// Mitsubishi GX Works2 project: BookEX6_40 String   PLC: Q13UDV

// global labels: Global
VAR_GLOBAL
  bVar0 AT M5000 : BOOL;
  abArray0 AT M5010 : ARRAY [0..49] OF BOOL;
  sStr0 AT D5000 : STRING[199];
  sStr1 AT D5100 : STRING[199];
  sStr2 AT D5200 : STRING[199];
  sStr3 AT D5300 : STRING[199];
  sStr4 AT D5400 : STRING[199];
  sStr5 AT D5500 : STRING[199];
  sStr6 AT D5600 : STRING[199];
  sStr7 AT D5700 : STRING[199];
  sStr8 AT D5800 : STRING[199];
  sStr9 AT D5900 : STRING[199];
  iVar0 AT D4500 : INT;
  iVar1 AT D4501 : INT;
  iVar2 AT D4502 : INT;
  iVar3 AT D4503 : INT;
  iVar4 AT D4504 : INT;
  iVar5 AT D4505 : INT;
  iVar6 AT D4506 : INT;
  iVar7 AT D4507 : INT;
  iVar8 AT D4508 : INT;
  iVar9 AT D4509 : INT;
  dVar0 AT D4510 : DINT;
  dVar1 AT D4512 : DINT;
  dVar2 AT D4514 : DINT;
  dVar3 AT D4516 : DINT;
  dVar4 AT D4518 : DINT;
  dVar5 AT D4520 : DINT;
  dVar6 AT D4522 : DINT;
  dVar7 AT D4524 : DINT;
  dVar8 AT D4526 : DINT;
  dVar9 AT D4528 : DINT;
  wVar0 AT D4530 : WORD;
  wVar1 AT D4531 : WORD;
  wVar2 AT D4532 : WORD;
  wVar3 AT D4533 : WORD;
  wVar4 AT D4534 : WORD;
  wVar5 AT D4535 : WORD;
  wVar6 AT D4536 : WORD;
  wVar7 AT D4537 : WORD;
  wVar8 AT D4538 : WORD;
  wVar9 AT D4539 : WORD;
  dwVar0 AT D4540 : DWORD;
  dwVar1 AT D4542 : DWORD;
  dwVar2 AT D4544 : DWORD;
  dwVar3 AT D4546 : DWORD;
  dwVar4 AT D4548 : DWORD;
  dwVar5 AT D4550 : DWORD;
  dwVar6 AT D4552 : DWORD;
  dwVar7 AT D4554 : DWORD;
  dwVar8 AT D4556 : DWORD;
  dwVar9 AT D4558 : DWORD;
  fsVar0 AT D4560 : REAL;
  fsVar1 AT D4562 : REAL;
  fsVar2 AT D4564 : REAL;
  fsVar3 AT D4566 : REAL;
  fsVar4 AT D4568 : REAL;
  fsVar5 AT D4570 : REAL;
  fsVar6 AT D4572 : REAL;
  fsVar7 AT D4574 : REAL;
  fsVar8 AT D4576 : REAL;
  fsVar9 AT D4578 : REAL;
  fdVar0 AT D4580 : LREAL;
  tTime0 AT D4620 : TIME;
  tTime1 AT D4622 : TIME;
  tTime2 AT D4624 : TIME;
  tTime3 AT D4626 : TIME;
  tTime4 AT D4628 : TIME;
  tTime5 AT D4630 : TIME;
  tTime6 AT D4632 : TIME;
  tTime7 AT D4634 : TIME;
  tTime8 AT D4636 : TIME;
  tTime9 AT D4638 : TIME;
  tTime10 AT D4640 : TIME;
  bVar1 AT M5001 : BOOL;
  bVar2 AT M5002 : BOOL;
  bVar3 AT M5003 : BOOL;
  bVar4 AT M5004 : BOOL;
  bVar5 AT M5005 : BOOL;
  bVar6 AT M5006 : BOOL;
  bVar7 AT M5007 : BOOL;
  bVar8 AT M5008 : BOOL;
  bVar9 AT M5009 : BOOL;
  abArray1 AT M5060 : ARRAY [0..49] OF BOOL;
  abArray2 AT M5110 : ARRAY [0..49] OF BOOL;
  abArray3 AT M5160 : ARRAY [0..49] OF BOOL;
  abArray4 AT M5210 : ARRAY [0..49] OF BOOL;
  abArray5 AT M5260 : ARRAY [0..49] OF BOOL;
  abArray6 AT M5310 : ARRAY [0..49] OF BOOL;
  abArray7 AT M5360 : ARRAY [0..49] OF BOOL;
  abArray8 AT M5410 : ARRAY [0..49] OF BOOL;
  abArray9 AT M5460 : ARRAY [0..49] OF BOOL;
  fdVar1 AT D4584 : LREAL;
  fdVar2 AT D4588 : LREAL;
  fdVar3 AT D4592 : LREAL;
  fdVar4 AT D4596 : LREAL;
  fdVar5 AT D4600 : LREAL;
  fdVar6 AT D4604 : LREAL;
  fdVar7 AT D4608 : LREAL;
  fdVar8 AT D4612 : LREAL;
  fdVar9 AT D4616 : LREAL;
  afsPen0 AT D2000 : ARRAY [0..499] OF REAL;
  afsPen1 AT D3000 : ARRAY [0..499] OF REAL;
  SpecStr AT D4999 : STRING[1];
  adwD10 AT D10 : ARRAY [0..9] OF DWORD;
  awD10 AT D10 : ARRAY [0..19] OF WORD;
  abM10 AT M10 : ARRAY [0..19] OF BOOL;
END_VAR
// user libraries (not included): HMI

PROGRAM ExASC_HEX
VAR
  Mov4WORD_1 : Mov4WORD;
  Mov4WORD_2 : Mov4WORD;
END_VAR
(* structured ladder/FBD written out as ST: instructions are called as NAME(EN, inputs, outputs); _pN, _eN, _tN stand for wires *)
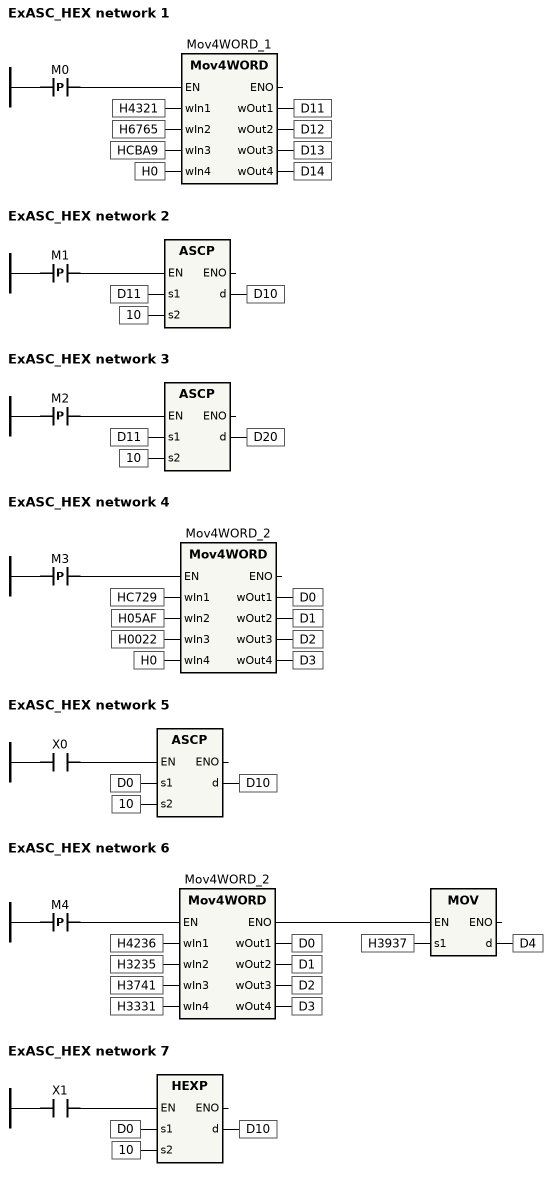
(* network 1 *)
Mov4WORD_1(EN := LDP(TRUE, M0), wIn1 := H4321, wIn2 := H6765, wIn3 := HCBA9, wIn4 := H0, wOut1 => D11, wOut2 => D12, wOut3 => D13, wOut4 => D14);
(* network 2 *)
ASCP(LDP(TRUE, M1), D11, 10, D10);
(* network 3 *)
ASCP(LDP(TRUE, M2), D11, 10, D20);
(* network 4 *)
Mov4WORD_2(EN := LDP(TRUE, M3), wIn1 := HC729, wIn2 := H05AF, wIn3 := H0022, wIn4 := H0, wOut1 => D0, wOut2 => D1, wOut3 => D2, wOut4 => D3);
(* network 5 *)
ASCP(X0, D0, 10, D10);
(* network 6 *)
Mov4WORD_2(EN := LDP(TRUE, M4), wIn1 := H4236, wIn2 := H3235, wIn3 := H3741, wIn4 := H3331, wOut1 => D0, wOut2 => D1, wOut3 => D2, wOut4 => D3);
MOV(Mov4WORD_2.ENO, H3937, D4);
(* network 7 *)
HEXP(X1, D0, 10, D10);
END_PROGRAM

PROGRAM ExBCDDA
VAR
  newBCDDA_1 : newBCDDA;
  sTemp : STRING[6];
END_VAR
(* structured ladder/FBD written out as ST: instructions are called as NAME(EN, inputs, outputs); _pN, _eN, _tN stand for wires *)
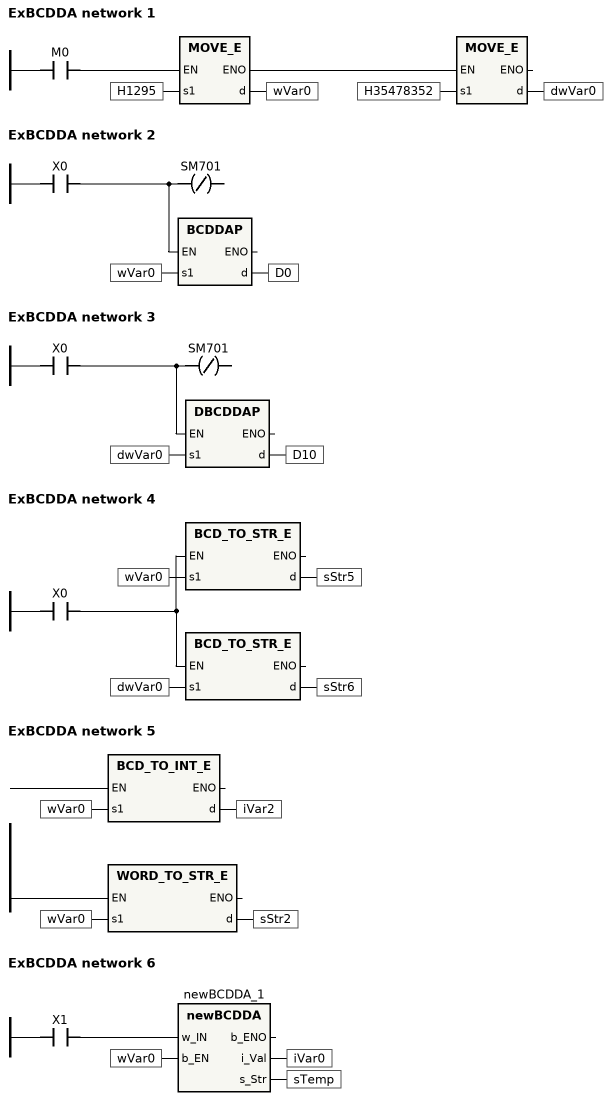
(* network 1 *)
_e1 := MOVE_E(M0, H1295, wVar0);
MOVE_E(_e1, H35478352, dwVar0);
(* network 2 *)
SM701 := NOT X0;
BCDDAP(X0, wVar0, D0);
(* network 3 *)
SM701 := NOT X0;
DBCDDAP(X0, dwVar0, D10);
(* network 4 *)
BCD_TO_STR_E(X0, wVar0, sStr5);
BCD_TO_STR_E(X0, dwVar0, sStr6);
(* network 5 *)
BCD_TO_INT_E(TRUE, wVar0, iVar2);
WORD_TO_STR_E(TRUE, wVar0, sStr2);
(* network 6 *)
newBCDDA_1(w_IN := X1, b_EN := wVar0, i_Val => iVar0, s_Str => sTemp);
END_PROGRAM

PROGRAM ExBINDA
(* structured ladder/FBD written out as ST: instructions are called as NAME(EN, inputs, outputs); _pN, _eN, _tN stand for wires *)
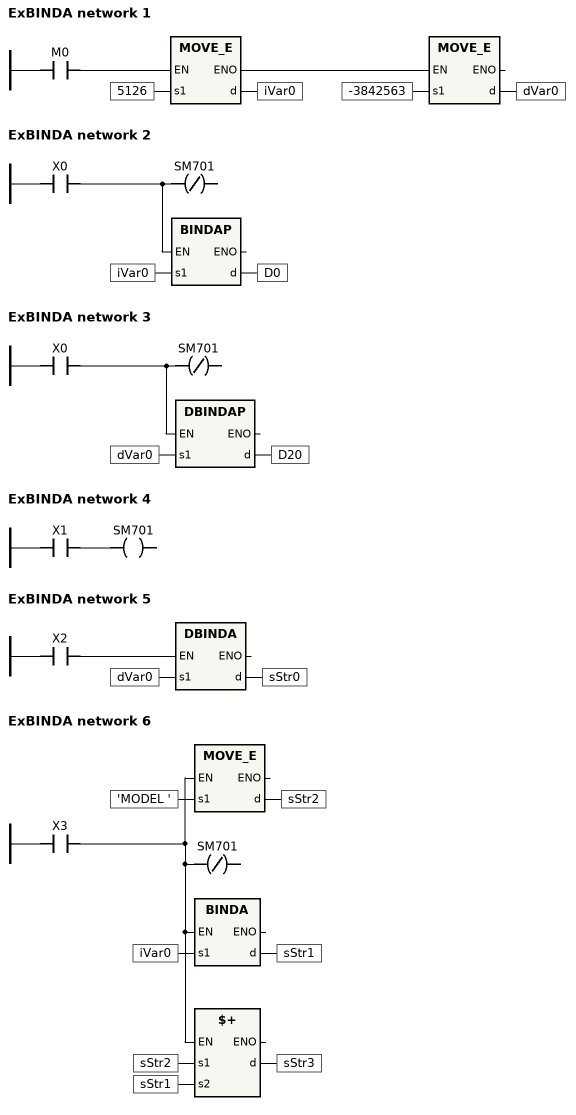
(* network 1 *)
_e1 := MOVE_E(M0, 5126, iVar0);
MOVE_E(_e1, -3842563, dVar0);
(* network 2 *)
SM701 := NOT X0;
BINDAP(X0, iVar0, D0);
(* network 3 *)
SM701 := NOT X0;
DBINDAP(X0, dVar0, D20);
(* network 4 *)
SM701 := X1;
(* network 5 *)
DBINDA(X2, dVar0, sStr0);
(* network 6 *)
SM701 := NOT X3;
MOVE_E(X3, 'MODEL ', sStr2);
BINDA(X3, iVar0, sStr1);
$+(X3, sStr2, sStr1, sStr3);
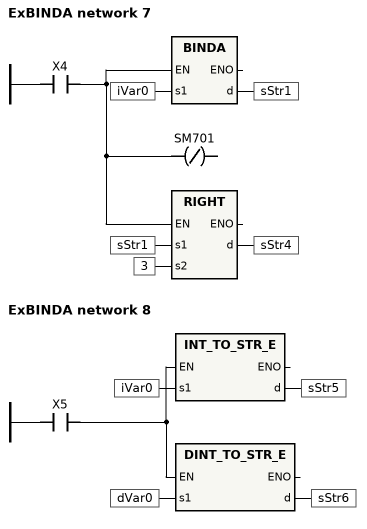
(* network 7 *)
SM701 := NOT X4;
BINDA(X4, iVar0, sStr1);
RIGHT(X4, sStr1, 3, sStr4);
(* network 8 *)
INT_TO_STR_E(X5, iVar0, sStr5);
DINT_TO_STR_E(X5, dVar0, sStr6);
END_PROGRAM

PROGRAM ExBINHA
VAR
  sStr40 : STRING[4];
  sStr41 : STRING[4];
END_VAR
(* structured ladder/FBD written out as ST: instructions are called as NAME(EN, inputs, outputs); _pN, _eN, _tN stand for wires *)
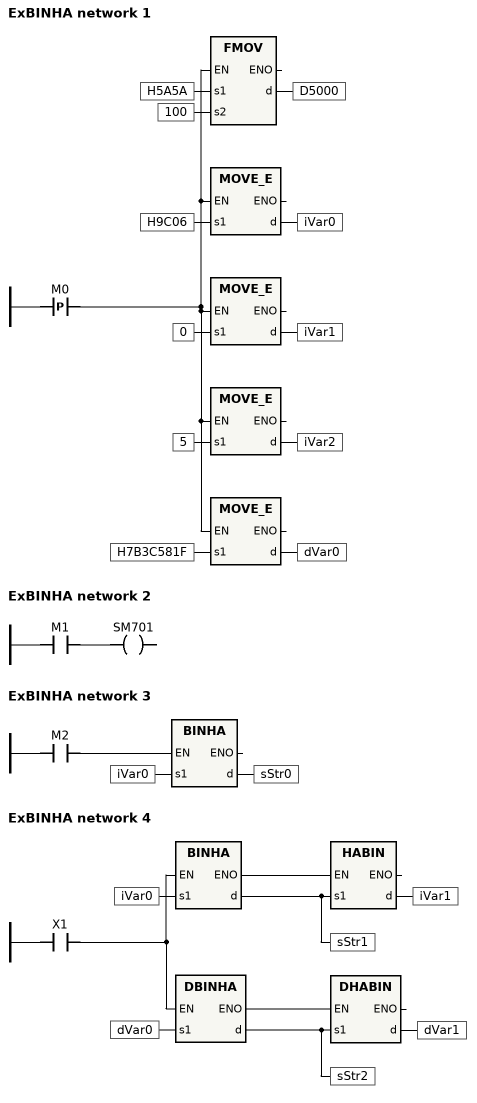
(* network 1 *)
_p1 := LDP(TRUE, M0);
FMOV(_p1, H5A5A, 100, D5000);
MOVE_E(_p1, H9C06, iVar0);
MOVE_E(_p1, 0, iVar1);
MOVE_E(_p1, 5, iVar2);
MOVE_E(_p1, H7B3C581F, dVar0);
(* network 2 *)
SM701 := M1;
(* network 3 *)
BINHA(M2, iVar0, sStr0);
(* network 4 *)
_e1 := BINHA(X1, iVar0, sStr1);
HABIN(_e1, sStr1, iVar1);
_e2 := DBINHA(X1, dVar0, sStr2);
DHABIN(_e2, sStr2, dVar1);
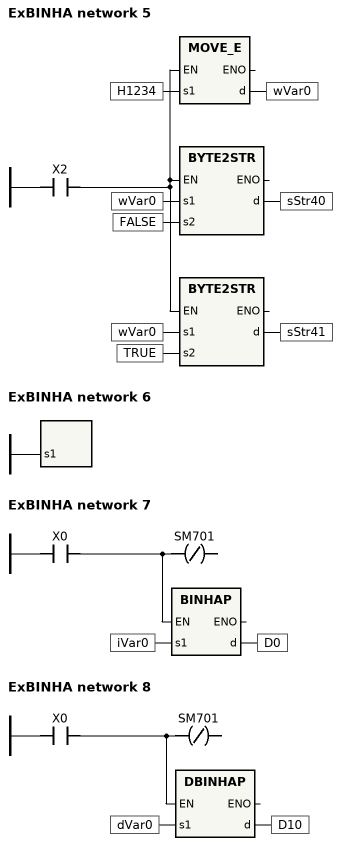
(* network 5 *)
MOVE_E(X2, H1234, wVar0);
BYTE2STR(X2, wVar0, FALSE, sStr40);
BYTE2STR(X2, wVar0, TRUE, sStr41);
(* network 6 *)
(* element kind 10  <- TRUE *)
(* network 7 *)
SM701 := NOT X0;
BINHAP(X0, iVar0, D0);
(* network 8 *)
SM701 := NOT X0;
DBINHAP(X0, dVar0, D10);
END_PROGRAM

PROGRAM ExCOMRD
VAR
  aiTmp : ARRAY [0..1] OF INT;
END_VAR
(* structured ladder/FBD written out as ST: instructions are called as NAME(EN, inputs, outputs); _pN, _eN, _tN stand for wires *)
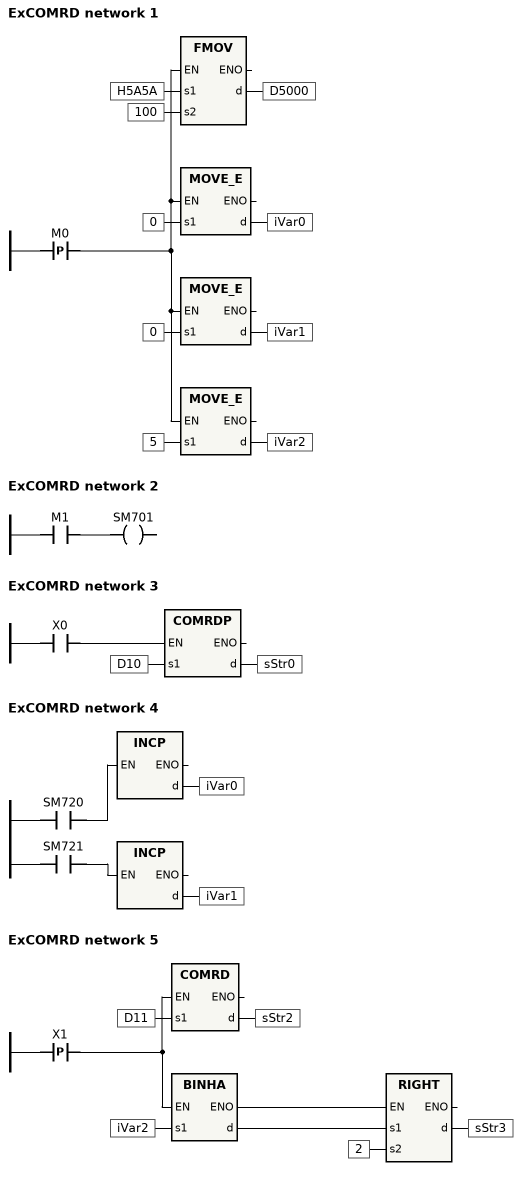
(* network 1 *)
_p1 := LDP(TRUE, M0);
FMOV(_p1, H5A5A, 100, D5000);
MOVE_E(_p1, 0, iVar0);
MOVE_E(_p1, 0, iVar1);
MOVE_E(_p1, 5, iVar2);
(* network 2 *)
SM701 := M1;
(* network 3 *)
COMRDP(X0, D10, sStr0);
(* network 4 *)
INCP(SM720, iVar0);
INCP(SM721, iVar1);
(* network 5 *)
_p1 := LDP(TRUE, X1);
COMRD(_p1, D11, sStr2);
_e3 := BINHA(_p1, iVar2, _t2);
RIGHT(_e3, _t2, 2, sStr3);
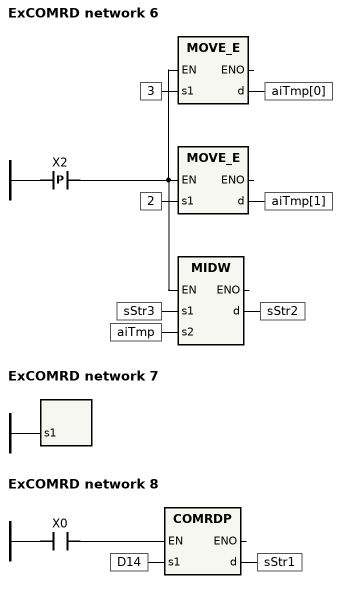
(* network 6 *)
_p1 := LDP(TRUE, X2);
MOVE_E(_p1, 3, aiTmp[0]);
MOVE_E(_p1, 2, aiTmp[1]);
MIDW(_p1, sStr3, aiTmp, sStr2);
(* network 7 *)
(* element kind 10  <- TRUE *)
(* network 8 *)
COMRDP(X0, D14, sStr1);
END_PROGRAM

PROGRAM ExDABCD
VAR
  UpperSTR_1 : UpperSTR;
  UpperSTR_2 : UpperSTR;
END_VAR
(* structured ladder/FBD written out as ST: instructions are called as NAME(EN, inputs, outputs); _pN, _eN, _tN stand for wires *)
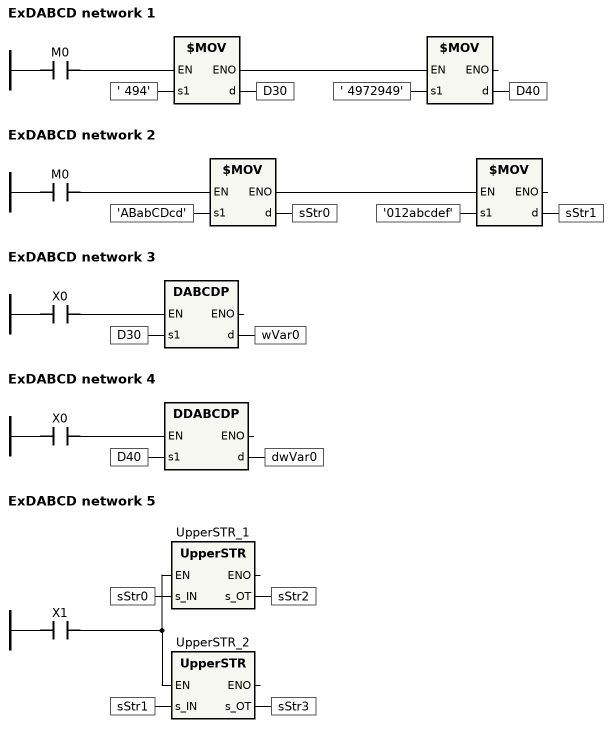
(* network 1 *)
_e1 := $MOV(M0, ' 494', D30);
$MOV(_e1, ' 4972949', D40);
(* network 2 *)
_e1 := $MOV(M0, 'ABabCDcd', sStr0);
$MOV(_e1, '012abcdef', sStr1);
(* network 3 *)
DABCDP(X0, D30, wVar0);
(* network 4 *)
DDABCDP(X0, D40, dwVar0);
(* network 5 *)
UpperSTR_1(EN := X1, s_IN := sStr0, s_OT => sStr2);
UpperSTR_2(EN := X1, s_IN := sStr1, s_OT => sStr3);
END_PROGRAM

PROGRAM ExDABIN
(* structured ladder/FBD written out as ST: instructions are called as NAME(EN, inputs, outputs); _pN, _eN, _tN stand for wires *)
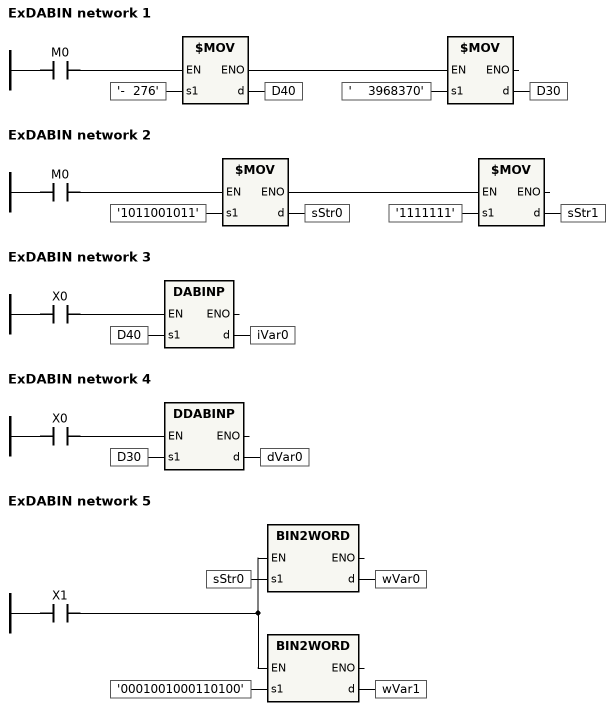
(* network 1 *)
_e1 := $MOV(M0, '-  276', D40);
$MOV(_e1, '    3968370', D30);
(* network 2 *)
_e1 := $MOV(M0, '1011001011', sStr0);
$MOV(_e1, '1111111', sStr1);
(* network 3 *)
DABINP(X0, D40, iVar0);
(* network 4 *)
DDABINP(X0, D30, dVar0);
(* network 5 *)
BIN2WORD(X1, sStr0, wVar0);
BIN2WORD(X1, '0001001000110100', wVar1);
END_PROGRAM

PROGRAM ExEMOD
VAR
  awBCD1 : ARRAY [0..4] OF WORD;
  Mov4WORD_1 : Mov4WORD;
  awBCD2 : ARRAY [0..4] OF WORD;
  awBCD3 : ARRAY [0..4] OF WORD;
  awBCD4 : ARRAY [0..4] OF WORD;
  Mov4WORD_2 : Mov4WORD;
  Mov4WORD_3 : Mov4WORD;
  Mov4WORD_4 : Mov4WORD;
  Mov4WORD_5 : Mov4WORD;
  awBCD5 : ARRAY [0..4] OF WORD;
  Mov4WORD_6 : Mov4WORD;
  awBCD6 : ARRAY [0..4] OF WORD;
END_VAR
(* structured ladder/FBD written out as ST: instructions are called as NAME(EN, inputs, outputs); _pN, _eN, _tN stand for wires *)
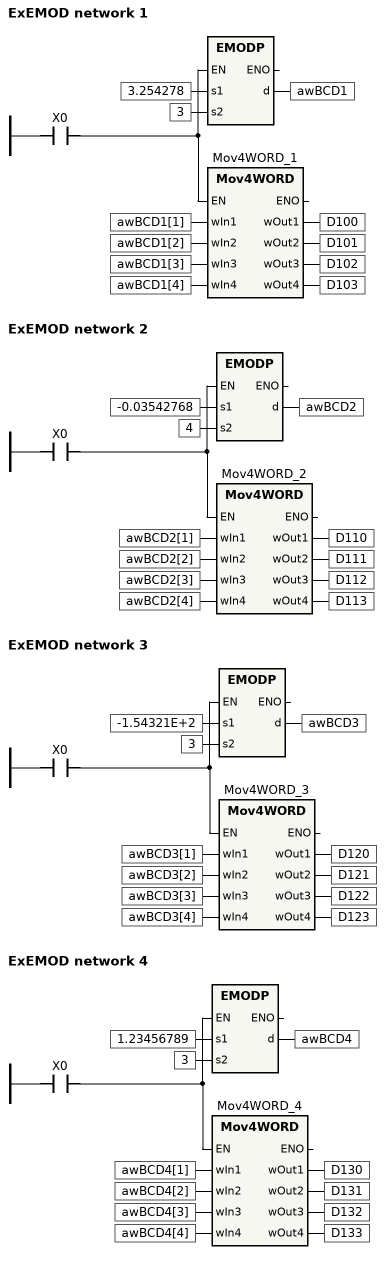
(* network 1 *)
EMODP(X0, 3.254278, 3, awBCD1);
Mov4WORD_1(EN := X0, wIn1 := awBCD1[1], wIn2 := awBCD1[2], wIn3 := awBCD1[3], wIn4 := awBCD1[4], wOut1 => D100, wOut2 => D101, wOut3 => D102, wOut4 => D103);
(* network 2 *)
EMODP(X0, -0.03542768, 4, awBCD2);
Mov4WORD_2(EN := X0, wIn1 := awBCD2[1], wIn2 := awBCD2[2], wIn3 := awBCD2[3], wIn4 := awBCD2[4], wOut1 => D110, wOut2 => D111, wOut3 => D112, wOut4 => D113);
(* network 3 *)
EMODP(X0, -1.54321E+2, 3, awBCD3);
Mov4WORD_3(EN := X0, wIn1 := awBCD3[1], wIn2 := awBCD3[2], wIn3 := awBCD3[3], wIn4 := awBCD3[4], wOut1 => D120, wOut2 => D121, wOut3 => D122, wOut4 => D123);
(* network 4 *)
EMODP(X0, 1.23456789, 3, awBCD4);
Mov4WORD_4(EN := X0, wIn1 := awBCD4[1], wIn2 := awBCD4[2], wIn3 := awBCD4[3], wIn4 := awBCD4[4], wOut1 => D130, wOut2 => D131, wOut3 => D132, wOut4 => D133);
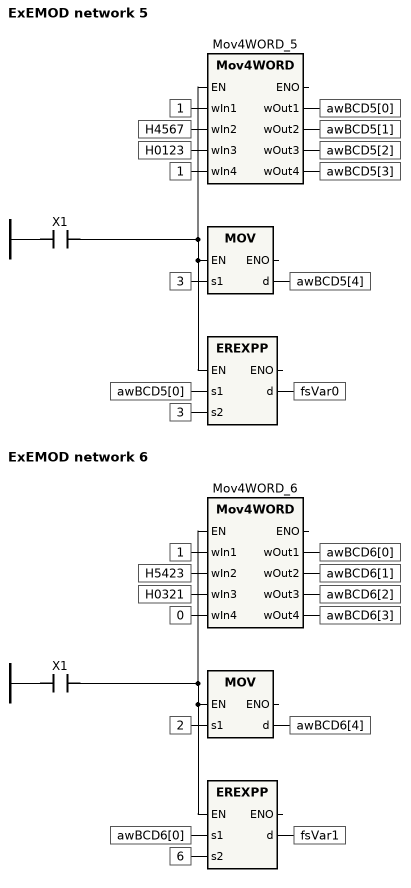
(* network 5 *)
Mov4WORD_5(EN := X1, wIn1 := 1, wIn2 := H4567, wIn3 := H0123, wIn4 := 1, wOut1 => awBCD5[0], wOut2 => awBCD5[1], wOut3 => awBCD5[2], wOut4 => awBCD5[3]);
MOV(X1, 3, awBCD5[4]);
EREXPP(X1, awBCD5[0], 3, fsVar0);
(* network 6 *)
Mov4WORD_6(EN := X1, wIn1 := 1, wIn2 := H5423, wIn3 := H0321, wIn4 := 0, wOut1 => awBCD6[0], wOut2 => awBCD6[1], wOut3 => awBCD6[2], wOut4 => awBCD6[3]);
MOV(X1, 2, awBCD6[4]);
EREXPP(X1, awBCD6[0], 6, fsVar1);
END_PROGRAM

PROGRAM ExHABIN
(* structured ladder/FBD written out as ST: instructions are called as NAME(EN, inputs, outputs); _pN, _eN, _tN stand for wires *)
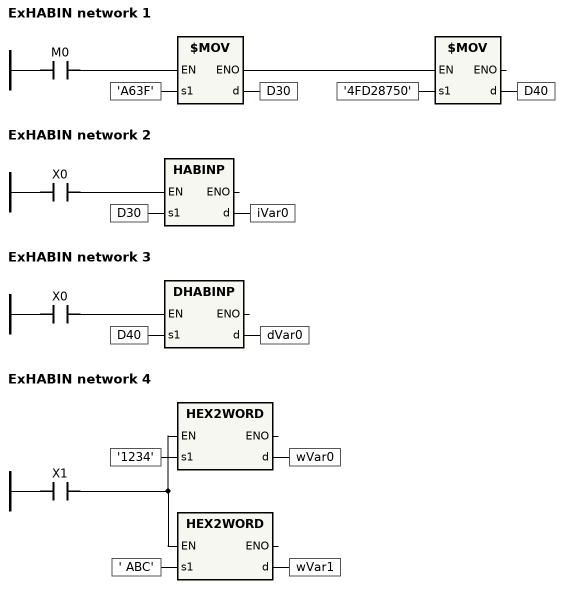
(* network 1 *)
_e1 := $MOV(M0, 'A63F', D30);
$MOV(_e1, '4FD28750', D40);
(* network 2 *)
HABINP(X0, D30, iVar0);
(* network 3 *)
DHABINP(X0, D40, dVar0);
(* network 4 *)
HEX2WORD(X1, '1234', wVar0);
HEX2WORD(X1, ' ABC', wVar1);
END_PROGRAM

PROGRAM ExLeftRight
(* structured ladder/FBD written out as ST: instructions are called as NAME(EN, inputs, outputs); _pN, _eN, _tN stand for wires *)
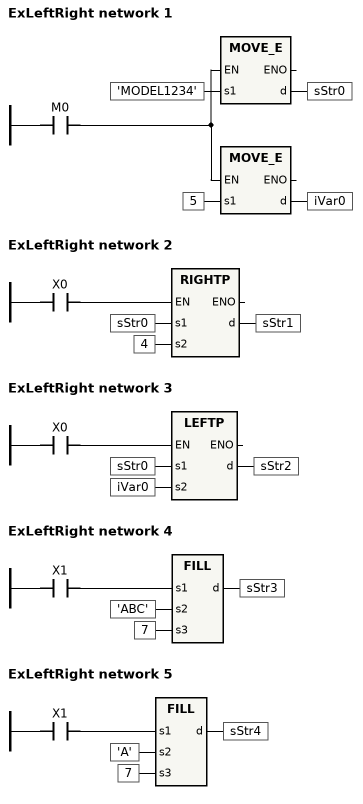
(* network 1 *)
MOVE_E(M0, 'MODEL1234', sStr0);
MOVE_E(M0, 5, iVar0);
(* network 2 *)
RIGHTP(X0, sStr0, 4, sStr1);
(* network 3 *)
LEFTP(X0, sStr0, iVar0, sStr2);
(* network 4 *)
sStr3 := FILL(X1, 'ABC', 7);
(* network 5 *)
sStr4 := FILL(X1, 'A', 7);
END_PROGRAM

PROGRAM ExLEN
(* structured ladder/FBD written out as ST: instructions are called as NAME(EN, inputs, outputs); _pN, _eN, _tN stand for wires *)
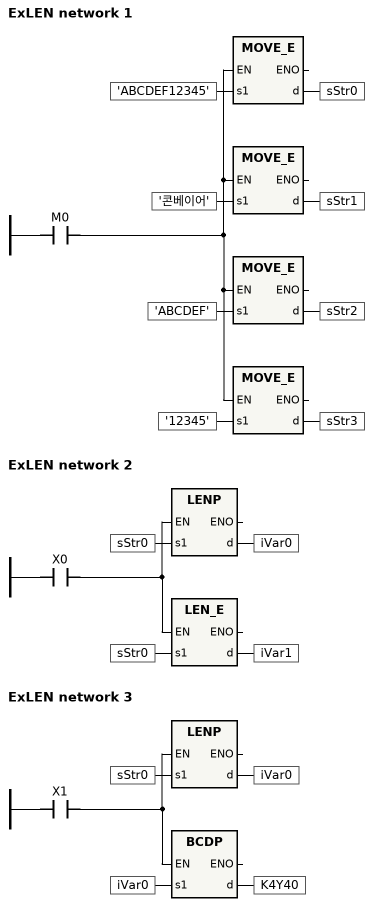
(* network 1 *)
MOVE_E(M0, 'ABCDEF12345', sStr0);
MOVE_E(M0, '콘베이어', sStr1);
MOVE_E(M0, 'ABCDEF', sStr2);
MOVE_E(M0, '12345', sStr3);
(* network 2 *)
LENP(X0, sStr0, iVar0);
LEN_E(X0, sStr0, iVar1);
(* network 3 *)
LENP(X1, sStr0, iVar0);
BCDP(X1, iVar0, K4Y40);
END_PROGRAM

PROGRAM ExMID
VAR
  aiVar0 : ARRAY [0..1] OF INT;
  aiVar1 : ARRAY [0..1] OF INT;
END_VAR
(* structured ladder/FBD written out as ST: instructions are called as NAME(EN, inputs, outputs); _pN, _eN, _tN stand for wires *)
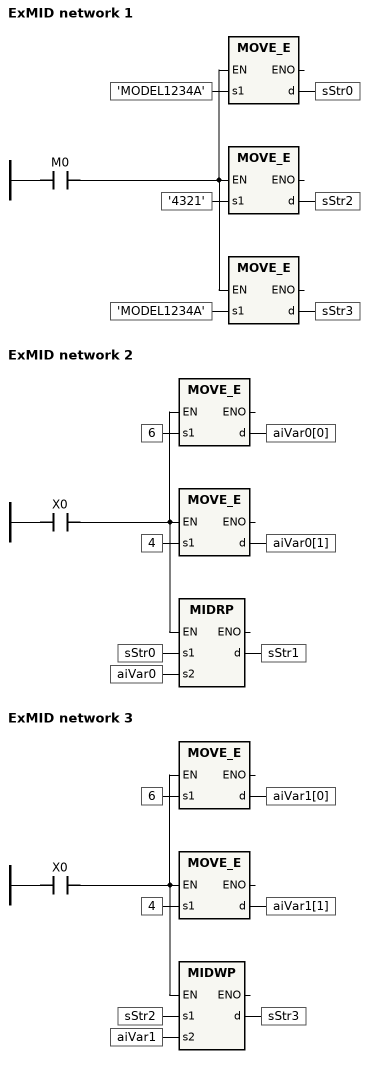
(* network 1 *)
MOVE_E(M0, 'MODEL1234A', sStr0);
MOVE_E(M0, '4321', sStr2);
MOVE_E(M0, 'MODEL1234A', sStr3);
(* network 2 *)
MOVE_E(X0, 6, aiVar0[0]);
MOVE_E(X0, 4, aiVar0[1]);
MIDRP(X0, sStr0, aiVar0, sStr1);
(* network 3 *)
MOVE_E(X0, 6, aiVar1[0]);
MOVE_E(X0, 4, aiVar1[1]);
MIDWP(X0, sStr2, aiVar1, sStr3);
END_PROGRAM

PROGRAM ExSTR
VAR
  aiVar3 : ARRAY [0..2] OF INT;
END_VAR
(* structured ladder/FBD written out as ST: instructions are called as NAME(EN, inputs, outputs); _pN, _eN, _tN stand for wires *)
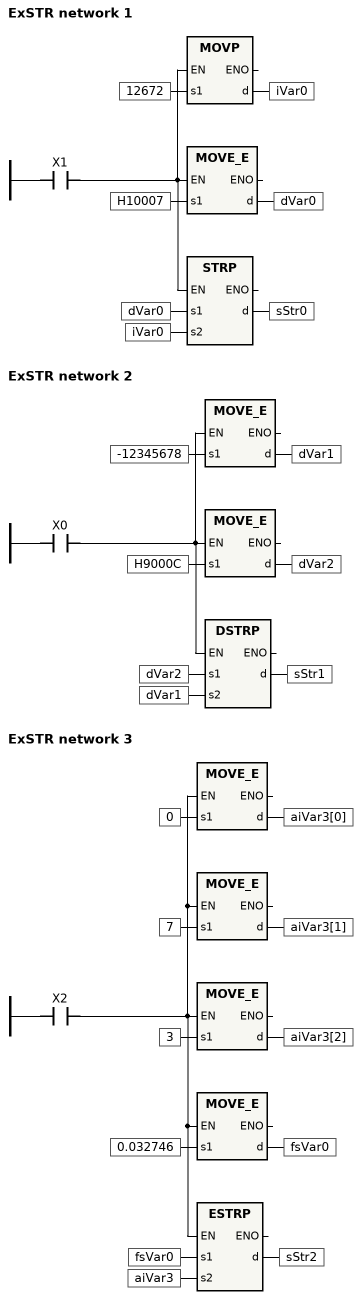
(* network 1 *)
MOVP(X1, 12672, iVar0);
MOVE_E(X1, H10007, dVar0);
STRP(X1, dVar0, iVar0, sStr0);
(* network 2 *)
MOVE_E(X0, -12345678, dVar1);
MOVE_E(X0, H9000C, dVar2);
DSTRP(X0, dVar2, dVar1, sStr1);
(* network 3 *)
MOVE_E(X2, 0, aiVar3[0]);
MOVE_E(X2, 7, aiVar3[1]);
MOVE_E(X2, 3, aiVar3[2]);
MOVE_E(X2, 0.032746, fsVar0);
ESTRP(X2, fsVar0, aiVar3, sStr2);
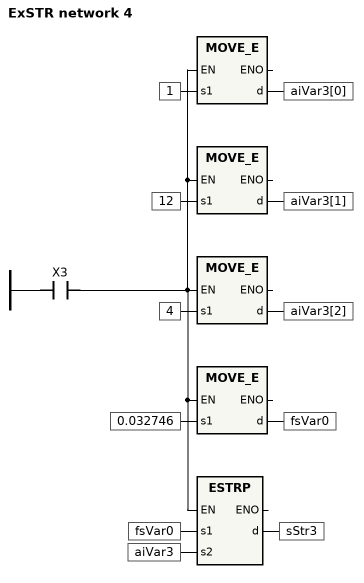
(* network 4 *)
MOVE_E(X3, 1, aiVar3[0]);
MOVE_E(X3, 12, aiVar3[1]);
MOVE_E(X3, 4, aiVar3[2]);
MOVE_E(X3, 0.032746, fsVar0);
ESTRP(X3, fsVar0, aiVar3, sStr3);
END_PROGRAM

PROGRAM ExString
VAR
  Var_D0 : WORD;
  Var_D1 : INT;
  sTmpStr1 : STRING[199];
  sTmpStr2 : STRING[199];
  sTmpStr3 : STRING[199];
  sTmpStr4 : STRING[199];
  sTmpStr5 : STRING[199];
  sTmpStr6 : STRING[199];
  sTmpStr7 : STRING[199];
  sTmpStr8 : STRING[199];
  sTmpStr9 : STRING[199];
  aiVar0 : ARRAY [0..1] OF INT;
  aiVar1 : ARRAY [0..1] OF INT;
END_VAR
(* structured ladder/FBD written out as ST: instructions are called as NAME(EN, inputs, outputs); _pN, _eN, _tN stand for wires *)
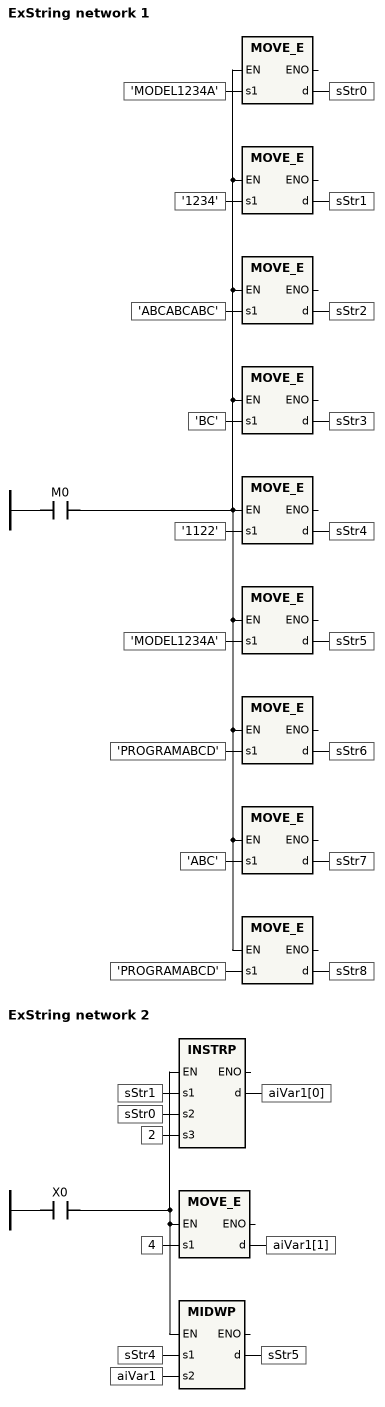
(* network 1 *)
MOVE_E(M0, 'MODEL1234A', sStr0);
MOVE_E(M0, '1234', sStr1);
MOVE_E(M0, 'ABCABCABC', sStr2);
MOVE_E(M0, 'BC', sStr3);
MOVE_E(M0, '1122', sStr4);
MOVE_E(M0, 'MODEL1234A', sStr5);
MOVE_E(M0, 'PROGRAMABCD', sStr6);
MOVE_E(M0, 'ABC', sStr7);
MOVE_E(M0, 'PROGRAMABCD', sStr8);
(* network 2 *)
INSTRP(X0, sStr1, sStr0, 2, aiVar1[0]);
MOVE_E(X0, 4, aiVar1[1]);
MIDWP(X0, sStr4, aiVar1, sStr5);
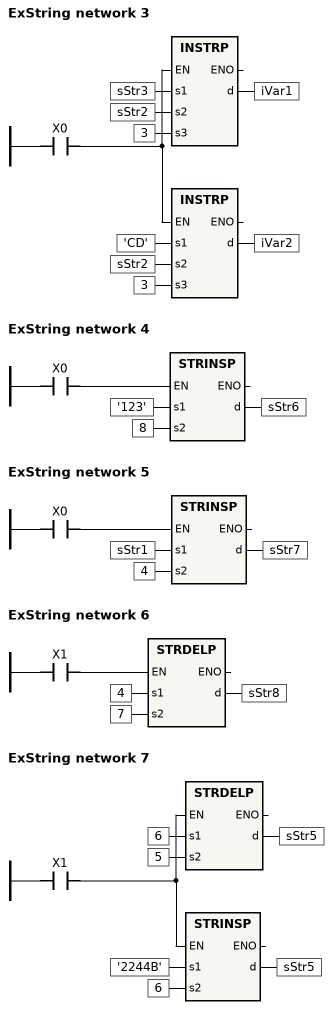
(* network 3 *)
INSTRP(X0, sStr3, sStr2, 3, iVar1);
INSTRP(X0, 'CD', sStr2, 3, iVar2);
(* network 4 *)
STRINSP(X0, '123', 8, sStr6);
(* network 5 *)
STRINSP(X0, sStr1, 4, sStr7);
(* network 6 *)
STRDELP(X1, 4, 7, sStr8);
(* network 7 *)
STRDELP(X1, 6, 5, sStr5);
STRINSP(X1, '2244B', 6, sStr5);
END_PROGRAM

PROGRAM ExVAL
VAR
  adVar0 : ARRAY [0..1] OF DINT;
  adVar1 : ARRAY [0..1] OF DINT;
END_VAR
(* structured ladder/FBD written out as ST: instructions are called as NAME(EN, inputs, outputs); _pN, _eN, _tN stand for wires *)
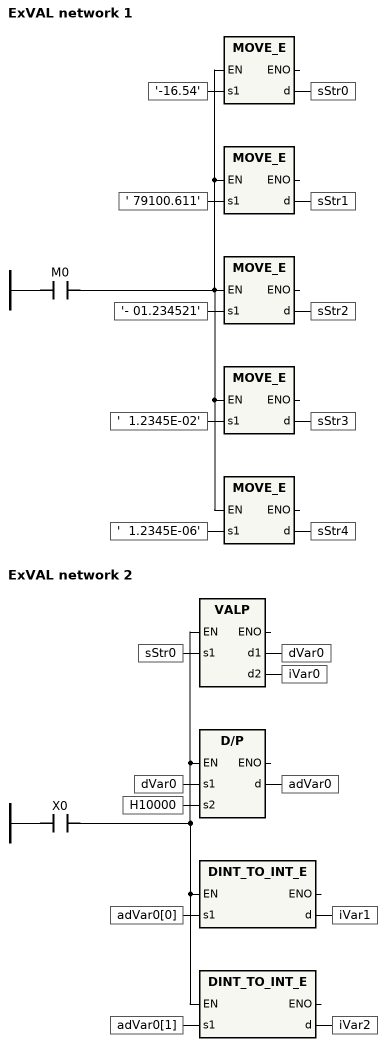
(* network 1 *)
MOVE_E(M0, '-16.54', sStr0);
MOVE_E(M0, ' 79100.611', sStr1);
MOVE_E(M0, '- 01.234521', sStr2);
MOVE_E(M0, '  1.2345E-02', sStr3);
MOVE_E(M0, '  1.2345E-06', sStr4);
(* network 2 *)
VALP(X0, sStr0, dVar0, iVar0);
D/P(X0, dVar0, H10000, adVar0);
DINT_TO_INT_E(X0, adVar0[0], iVar1);
DINT_TO_INT_E(X0, adVar0[1], iVar2);
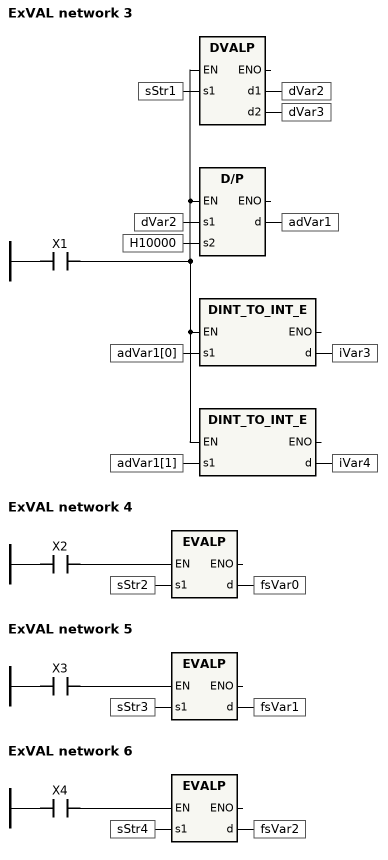
(* network 3 *)
DVALP(X1, sStr1, dVar2, dVar3);
D/P(X1, dVar2, H10000, adVar1);
DINT_TO_INT_E(X1, adVar1[0], iVar3);
DINT_TO_INT_E(X1, adVar1[1], iVar4);
(* network 4 *)
EVALP(X2, sStr2, fsVar0);
(* network 5 *)
EVALP(X3, sStr3, fsVar1);
(* network 6 *)
EVALP(X4, sStr4, fsVar2);
END_PROGRAM

FUNCTION BIN2WORD
VAR_INPUT
  s_IN : STRING[199];
END_VAR
VAR
  ix : INT;
  iLeng : INT;
  iChar : INT;
  sTmpStr : STRING[199];
  wTmp : WORD;
END_VAR
;
sTmpStr := s_IN;
LEN_E(TRUE, s_IN, iLeng);
IF iLeng = 0 THEN
	BIN2WORD := 0;
	RETURN;
END_IF;
wTmp := 0;
FOR ix := 1 TO iLeng DO
	iChar := GET_INT_ADDR(sTmpStr) MOD 256;
	IF iChar = 48 THEN
		wTmp := SHL(wTmp,1);
	ELSIF iChar = 49 THEN
		wTmp := SHL(wTmp,1) OR H0001;
	END_IF;
	sTmpStr := DELETE(sTmpStr, 1, 1);
END_FOR;
BIN2WORD := wTmp;
END_FUNCTION

FUNCTION BYTE2STR
VAR_INPUT
  w_IN : WORD;
END_VAR
VAR
  sTmpStr1 : STRING[4];
  wTmp : WORD;
END_VAR
VAR_INPUT
  b_HI : BOOL;
END_VAR
VAR
  sTmpStr2 : STRING[6];
END_VAR
;
wTmp := w_IN;
IF b_HI THEN
	wTmp := SHR(wTmp, 8);
END_IF;
wTmp := wTmp AND H00FF;
BINHA(TRUE, wTmp, sTmpStr2);
RIGHT(TRUE, sTmpStr2, 2, sTmpStr1);
BYTE2STR := sTmpStr1;
END_FUNCTION

FUNCTION FILL
VAR_INPUT
  b_EN : BOOL;
  s_Str : STRING[32];
END_VAR
VAR
  ix : INT;
END_VAR
VAR_INPUT
  i_Len : INT;
END_VAR
VAR
  sTemp : STRING[199];
END_VAR
;
LEN(TRUE, s_Str, ix);
IF NOT b_EN OR (i_Len*ix) > 199 THEN
	FILL := '';
	RETURN;
END_IF;
sTemp := '';
FOR ix := 1 TO i_Len DO
	sTemp := CONCAT(sTemp,s_Str);
END_FOR;
FILL := sTemp;
END_FUNCTION

FUNCTION HEX2WORD
VAR_INPUT
  s_IN : STRING[199];
END_VAR
VAR
  ix : INT;
  iLeng : INT;
  iChar : INT;
  sTmpStr : STRING[199];
  iy : INT;
  wTmp : WORD;
END_VAR
;
sTmpStr := s_IN;
LEN_E(TRUE, s_IN, iLeng);
IF iLeng = 0 THEN
	HEX2WORD := 0;
	RETURN;
END_IF;
iy := MAXIMUM(4, iLeng);
wTmp := 0;
FOR ix := 1 TO iy DO
	iChar := GET_INT_ADDR(sTmpStr) MOD 256;
	IF iChar > 47 AND iChar < 58 THEN
		wTmp := SHL(wTmp,4) OR (INT_TO_WORD(iChar) AND H0000F);
	ELSIF iChar > 64 AND iChar < 71 THEN
		wTmp := SHL(wTmp,4) OR INT_TO_WORD(iChar - 55);
	ELSIF iChar > 96 AND iChar < 103 THEN
		wTmp := SHL(wTmp,4) OR INT_TO_WORD(iChar - 87);
	END_IF;
	sTmpStr := DELETE(sTmpStr, 1, 1);
END_FOR;
HEX2WORD := wTmp;
END_FUNCTION

FUNCTION_BLOCK newBCDDA
VAR_INPUT
  w_IN : WORD;
  b_EN : BOOL;
END_VAR
VAR_OUTPUT
  b_ENO : BOOL;
  i_Val : INT;
  s_Str : STRING[6];
END_VAR
VAR
  sTemp : STRING[6];
END_VAR
;
b_ENO := b_EN;
IF NOT b_EN THEN
	RETURN;
END_IF;
i_Val := BCD_TO_INT(w_IN);
sTemp := WORD_TO_STR(w_IN);
s_Str := sTemp;
END_FUNCTION_BLOCK

FUNCTION_BLOCK UpperSTR
VAR_INPUT
  s_IN : STRING[199];
END_VAR
VAR
  ix : INT;
  iChar : INT;
  iLeng : INT;
  wTmp : WORD;
  sTmpStr1 : STRING[199];
  sTmpStr2 : STRING[199];
END_VAR
VAR_OUTPUT
  s_OT : STRING[199];
END_VAR
;
sTmpStr1 := s_IN;
sTmpStr2 := '';
LEN_E(TRUE, s_IN, iLeng);
IF iLeng = 0 THEN
	s_OT:= sTmpStr2;
	RETURN;
END_IF;
FOR ix := 1 TO iLeng DO
	iChar := GET_INT_ADDR(sTmpStr1) MOD 256;
	IF iChar > 96 AND iChar < 123 THEN
		iChar := iChar - 32;
	END_IF;
	D4999 := iChar;
	sTmpStr1 := DELETE(sTmpStr1, 1, 1);
	sTmpStr2 := CONCAT(sTmpStr2, SpecStr);
END_FOR;
s_OT := sTmpStr2;
END_FUNCTION_BLOCK

FUNCTION UpperSTR2
VAR_INPUT
  s_IN : STRING[199];
END_VAR
VAR
  ix : INT;
  iLeng : INT;
  iChar : INT;
  sTmpStr1 : STRING[199];
  wTmp : WORD;
  sTmpStr2 : STRING[199];
END_VAR
;
sTmpStr1 := s_IN;
sTmpStr2 := '';
LEN_E(TRUE, s_IN, iLeng);
IF iLeng = 0 THEN
	UpperSTR := sTmpStr2;
	RETURN;
END_IF;
FOR ix := 1 TO iLeng DO
	iChar := GET_INT_ADDR(sTmpStr1) MOD 256;
	IF iChar > 96 AND iChar < 123 THEN
		iChar := iChar - 32;
	END_IF;
	D4999 := iChar;
	sTmpStr1 := DELETE(sTmpStr1, 1, 1);
	sTmpStr2 := CONCAT(sTmpStr2, D4999);
END_FOR;
UpperSTR := sTmpStr2;
END_FUNCTION

FUNCTION_BLOCK Split
VAR_INPUT
  bEN : BOOL;
  sDelimiter : STRING[9];
END_VAR
VAR_OUTPUT
  iLen : INT;
  sOut0 : STRING[199];
  sOut1 : STRING[199];
  sOut2 : STRING[199];
  sOut3 : STRING[199];
END_VAR
VAR_INPUT
  sInput : STRING[199];
END_VAR
VAR_OUTPUT
  bENO : BOOL;
  iCount : INT;
END_VAR
VAR
  Count : INT;
  ix : INT;
  iy : INT;
  aiPos : ARRAY [0..7] OF INT;
  asStr : ARRAY [0..7] OF STRING[199] := [8('')];
  aParam : ARRAY [0..1] OF INT;
END_VAR
;
IF LDP(TRUE, bEN) THEN
	LEN(TRUE, sInput, iLen);
	FOR  ix := 0 TO 7 DO 
		aiPos[ix] := 0;
		asStr[ix] := '';
	END_FOR;
	Count := 0;
	ix := 1;		iy := 0;
	WHILE ix < iLen AND Count < 8 AND iy = 0 DO
		INSTR(TRUE, sDelimiter, sInput, ix, aiPos[Count]);
		IF aiPos[Count] = 0 THEN 
			iy := 1; 
			aiPos[Count] := iLen + 1;
		ELSE
			ix := aiPos[Count] + 1;
			Count := Count + 1;
		END_IF;
	END_WHILE; 
	
	FOR  ix := 0 TO Count DO 
		IF ix = 0 THEN
			aParam[0] := 1;								(* Position *)
			aParam[1] := aiPos[ix] - 1;			(* No of Char *)
		ELSE
			aParam[0] := aiPos[ix-1] + 1;							(* Position *)
			aParam[1] := aiPos[ix] - aiPos[ix-1] - 1;		(* No of Char *)
		END_IF;	
		MIDR(TRUE, sInput, aParam, asStr[ix]);
	END_FOR;
END_IF;

sOut0 := asStr[0];
sOut1 := asStr[1];
sOut2 := asStr[2];
sOut3 := asStr[3];
iCount := Count + 1;
END_FUNCTION_BLOCK

PROGRAM ExSplit
VAR
  Split_1 : Split;
  Split_2 : Split;
  ssStr0 : STRING[199];
  ssStr1 : STRING[199];
  ssStr2 : STRING[199];
  ssStr3 : STRING[199];
  ssStr4 : STRING[199];
  ssStr5 : STRING[199];
  ssStr6 : STRING[199];
  ssStr7 : STRING[199];
  ssStr8 : STRING[199];
  bCmd : BOOL;
  ssStr9 : STRING[199];
END_VAR
(* structured ladder/FBD written out as ST: instructions are called as NAME(EN, inputs, outputs); _pN, _eN, _tN stand for wires *)
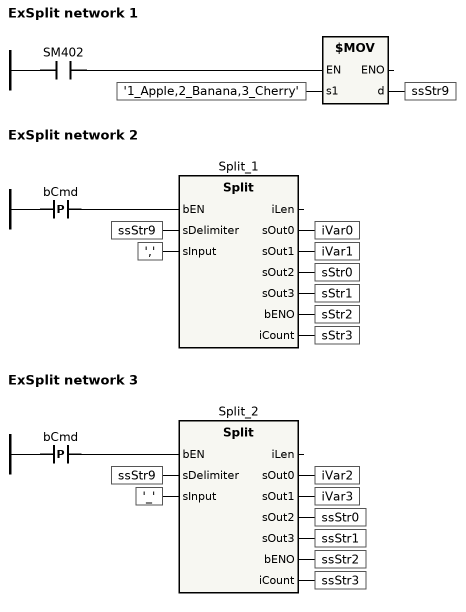
(* network 1 *)
$MOV(SM402, '1_Apple,2_Banana,3_Cherry', ssStr9);
(* network 2 *)
Split_1(bEN := LDP(TRUE, bCmd), sDelimiter := ssStr9, sInput := ',', sOut0 => iVar0, sOut1 => iVar1, sOut2 => sStr0, sOut3 => sStr1, bENO => sStr2, iCount => sStr3);
(* network 3 *)
Split_2(bEN := LDP(TRUE, bCmd), sDelimiter := ssStr9, sInput := '_', sOut0 => iVar2, sOut1 => iVar3, sOut2 => ssStr0, sOut3 => ssStr1, bENO => ssStr2, iCount => ssStr3);
END_PROGRAM
